// Mitsubishi GX Works2 project: ChuongTrinhMitshu1605202444444   PLC: FX1N/FX1NC

PROGRAM MAIN
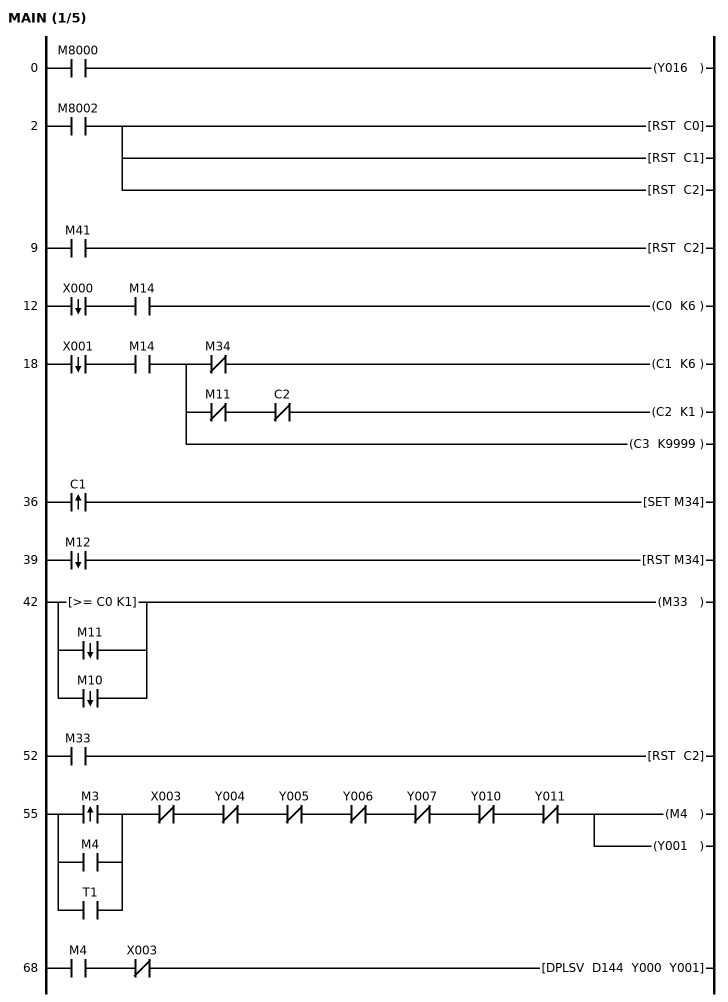
0     LD      M8000
      OUT     Y016
2     LD      M8002
      RST     C0
      RST     C1
      RST     C2
9     LD      M41
      RST     C2
12    LDF     X000
      AND     M14
      OUT     C0 K6
18    LDF     X001
      AND     M14
      MPS
      ANI     M34
      OUT     C1 K6
      MRD
      ANI     M11
      ANI     C2
      OUT     C2 K1
      MPP
      OUT     C3 K9999
36    LDP     C1
      SET     M34
39    LDF     M12
      RST     M34
42    LD>=    C0 K1
      ORF     M11
      ORF     M10
      OUT     M33
52    LD      M33
      RST     C2
55    LDP     M3
      OR      M4
      OR      T1
      ANI     X003
      ANI     Y004
      ANI     Y005
      ANI     Y006
      ANI     Y007
      ANI     Y010
      ANI     Y011
      OUT     M4
      OUT     Y001
68    LD      M4
      ANI     X003
      DPLSV   D144 Y000 Y001
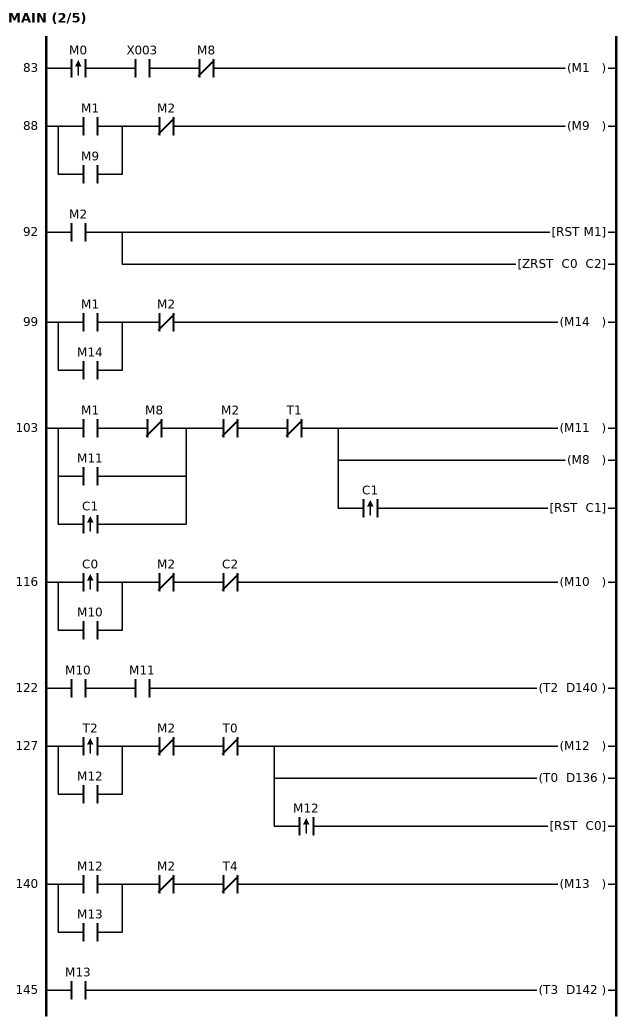
83    LDP     M0
      AND     X003
      ANI     M8
      OUT     M1
88    LD      M1
      OR      M9
      ANI     M2
      OUT     M9
92    LD      M2
      RST     M1
      ZRST    C0 C2
99    LD      M1
      OR      M14
      ANI     M2
      OUT     M14
103   LD      M1
      ANI     M8
      OR      M11
      ORP     C1
      ANI     M2
      ANI     T1
      OUT     M11
      OUT     M8
      ANDP    C1
      RST     C1
116   LDP     C0
      OR      M10
      ANI     M2
      ANI     C2
      OUT     M10
122   LD      M10
      AND     M11
      OUT     T2 D140
127   LDP     T2
      OR      M12
      ANI     M2
      ANI     T0
      OUT     M12
      OUT     T0 D136
      ANDP    M12
      RST     C0
140   LD      M12
      OR      M13
      ANI     M2
      ANI     T4
      OUT     M13
145   LD      M13
      OUT     T3 D142
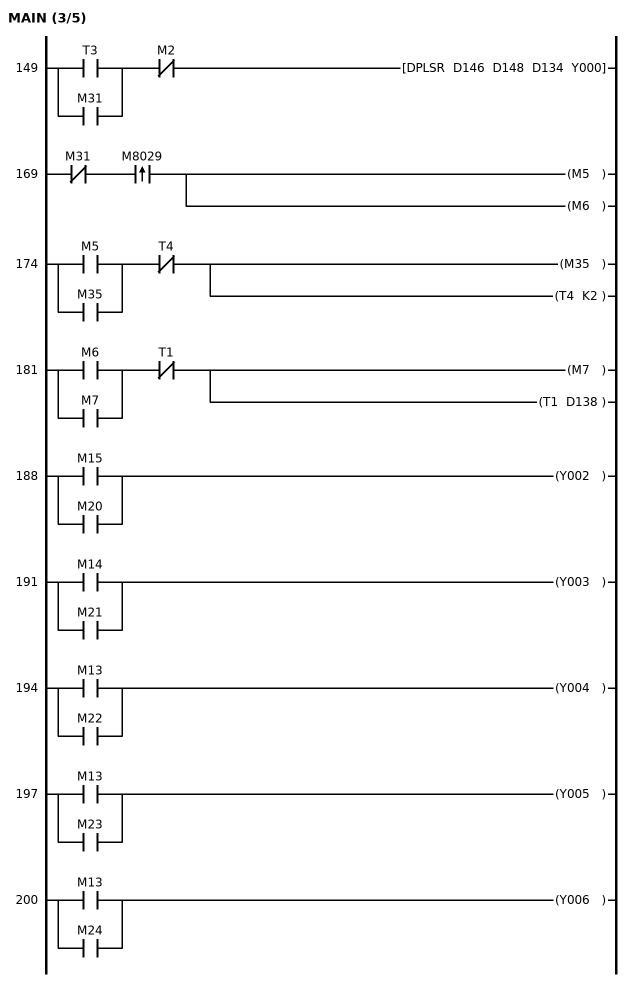
149   LD      T3
      OR      M31
      ANI     M2
      DPLSR   D146 D148 D134 Y000
169   LDI     M31
      ANDP    M8029
      OUT     M5
      OUT     M6
174   LD      M5
      OR      M35
      ANI     T4
      OUT     M35
      OUT     T4 K2
181   LD      M6
      OR      M7
      ANI     T1
      OUT     M7
      OUT     T1 D138
188   LD      M15
      OR      M20
      OUT     Y002
191   LD      M14
      OR      M21
      OUT     Y003
194   LD      M13
      OR      M22
      OUT     Y004
197   LD      M13
      OR      M23
      OUT     Y005
200   LD      M13
      OR      M24
      OUT     Y006
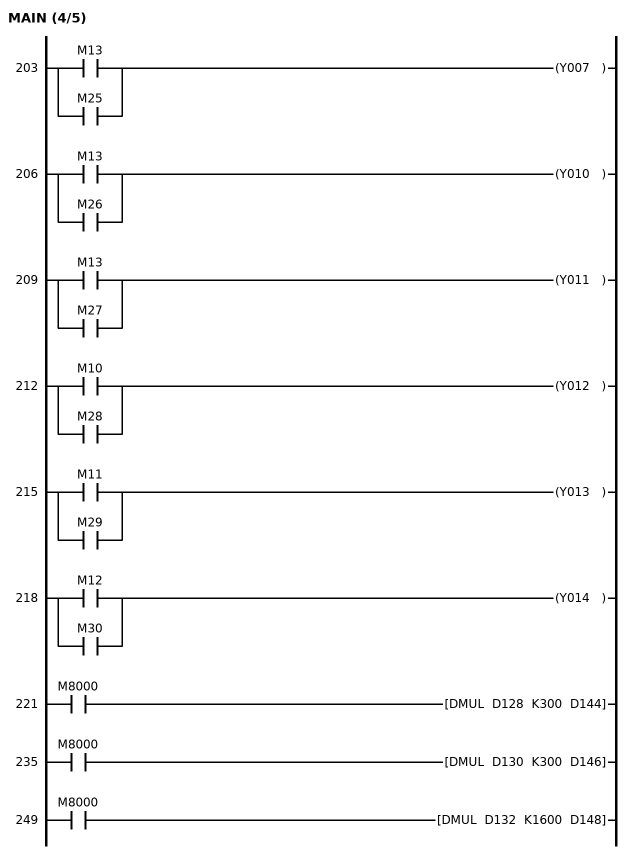
203   LD      M13
      OR      M25
      OUT     Y007
206   LD      M13
      OR      M26
      OUT     Y010
209   LD      M13
      OR      M27
      OUT     Y011
212   LD      M10
      OR      M28
      OUT     Y012
215   LD      M11
      OR      M29
      OUT     Y013
218   LD      M12
      OR      M30
      OUT     Y014
221   LD      M8000
      DMUL    D128 K300 D144
235   LD      M8000
      DMUL    D130 K300 D146
249   LD      M8000
      DMUL    D132 K1600 D148
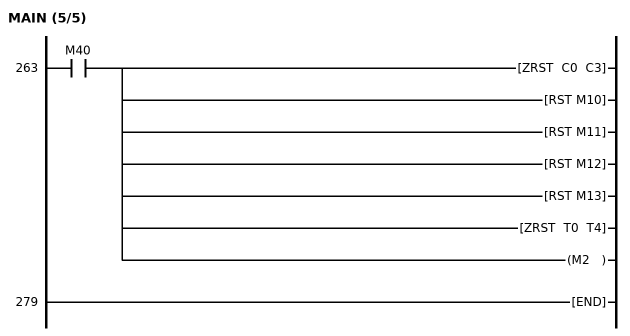
263   LD      M40
      ZRST    C0 C3
      RST     M10
      RST     M11
      RST     M12
      RST     M13
      ZRST    T0 T4
      OUT     M2
279   END
END_PROGRAM
